// Mitsubishi GX Works2 project: testCode   PLC: FX3G

// global labels: Global1
VAR_GLOBAL
  Jog_Left AT X004 : BOOL;
  Jog_Right AT X006 : BOOL;
  RelayMXC_1 AT Y001 : BOOL;
  RelayMXC_2 AT Y002 : BOOL;
  CommandMXC_F : BOOL;
  CommandMXC_R : BOOL;
  MXC_FWD : BOOL;
  MXC_Z : BOOL;
END_VAR
VAR_GLOBAL CONSTANT
  Round_MXC : REAL := 2.5;
END_VAR
VAR_GLOBAL
  Real_MXC : REAL;
  ModeAuto : BOOL;
  HSC AT C238 : DINT;
END_VAR
VAR_GLOBAL CONSTANT
  Speed_MXC : REAL := 1.5;
END_VAR
VAR_GLOBAL
  Freq_MXC : REAL;
  Round_Int : DWORD;
  Freq_Int : DWORD;
END_VAR

// task Task_01 (event TRUE, interval 0, priority 31): Control
// task InterruptMXC_Z (event I401, interval 0, priority 31): PickupX004

PROGRAM Control
VAR
  MXC : MotorRev;
  FlashF : R_TRIG;
  FlashZ : F_TRIG;
  PushOilPump : BOOL;
  ButtonOilP : BOOL;
  FlashP : R_TRIG;
  CounterCK : INT;
  Servo_MXC : Servo;
END_VAR
(* Khai bao vong quay cho MXC*)
EI( TRUE );
DEMUL( TRUE, E2000.0, Round_MXC , Real_MXC);
DEMUL(TRUE, E48000.0, Speed_MXC, Freq_MXC);
DINT( TRUE ,  Real_MXC , Round_Int );
DINT( TRUE ,  Freq_MXC , Freq_Int );
(*
MXC(SetAutoMan:= ModeAuto,
			LimitInputF := MXC_FWD , LimitInputR := MXC_Z,
			SetAutoRunF := CommandMXC_F, SetAutoRunR := CommandMXC_R,
			OutputF := RelayMXC_1, OutputR := RelayMXC_2);

RST( LDF(TRUE, MXC_FWD), M8054);
SET( LDF(TRUE, MXC_FWD), MXC_Z);
SET( LDF(TRUE, MXC_FWD), CommandMXC_R);
SET( CommandMXC_F AND X004, MXC_FWD);
RST( LDP(TRUE, CommandMXC_F), C251);

OUT_C_32( TRUE, CC251, K2147483647);
DHSCR( TRUE , REAL_TO_DINT( Real_MXC ), CN251, MXC_FWD);
 *)


Servo_MXC(SetAutoMan := ModeAuto,
						LimitInputF:= MXC_FWD, LimitInputR:= MXC_Z,
						Speed:=  Round_Int, Range:= Freq_Int,
						SetAutoRunF:= CommandMXC_F , SetAutoRunR:= CommandMXC_R ,
						OutputPLS:= Y0, OutputDIR:= Y4 );

RST( LDF(TRUE, MXC_FWD), M8054);
SET( LDF(TRUE, MXC_FWD), MXC_Z);
SET( LDF(TRUE, MXC_FWD), CommandMXC_R);
SET( CommandMXC_F AND X004, MXC_FWD);
RST( LDF(TRUE, M8340), MXC_FWD);




ButtonOilP := LDP(TRUE, PushOilPump) XOR ButtonOilP;
END_PROGRAM

FUNCTION_BLOCK MotorRev
VAR_INPUT
  SetAutoMan : BOOL;
END_VAR
VAR_IN_OUT
  PushManF : BOOL;
  PushManR : BOOL;
END_VAR
VAR_INPUT
  LimitInputF : BOOL;
  LimitInputR : BOOL;
END_VAR
VAR_IN_OUT
  SetAutoRunF : BOOL;
  SetAutoRunR : BOOL;
END_VAR
VAR_OUTPUT
  OutputF : BOOL;
  OutputR : BOOL;
END_VAR
VAR
  RelayBufferF : BOOL;
  RelayBufferR : BOOL;
END_VAR
(* Set mode Auto/Man *)
IF  SetAutoMan THEN
	RelayBufferF := 	NOT SetAutoRunR AND SetAutoRunF;
	RelayBufferR := NOT SetAutoRunF AND SetAutoRunR;
ELSE
	RelayBufferF := NOT PushManR AND PushManF;
	RelayBufferR := NOT PushManF AND PushManR;
END_IF;

OutputF := RelayBufferF AND LimitInputF ;
OutputR := RelayBufferR AND LimitInputR ;
(* Reset control signal *)
RST( LDF( TRUE, LimitInputF ) , RelayBufferF );
RST( LDF( TRUE, LimitInputF ) , SetAutoRunF );

RST( LDF( TRUE, LimitInputR ) , RelayBufferR );	
RST( LDF( TRUE, LimitInputR ) , SetAutoRunR );
END_FUNCTION_BLOCK

PROGRAM PickupX004
RST( TRUE, MXC_Z);
SET( TRUE, M8054);
END_PROGRAM

FUNCTION_BLOCK Servo
VAR_INPUT
  SetAutoMan : BOOL;
  LimitInputF : BOOL;
  LimitInputR : BOOL;
END_VAR
VAR_IN_OUT
  PushManF : BOOL;
  PushManR : BOOL;
END_VAR
VAR_INPUT
  Speed : DWORD;
  Range : DWORD;
END_VAR
VAR_IN_OUT
  SetAutoRunF : BOOL;
  SetAutoRunR : BOOL;
END_VAR
VAR_OUTPUT
  OutputPLS : BOOL;
  OutputDIR : BOOL;
END_VAR
VAR
  RelayPLS : BOOL;
  RelayDIR : BOOL;
END_VAR
(* Set mode Auto/Man *)
IF  SetAutoMan THEN
	RelayDIR := SetAutoRunR;
	RelayPLS := SetAutoRunF XOR SetAutoRunR;
ELSE
	RelayDIR := PushManR;
	RelayPLS := PushManF XOR PushManR;
END_IF;

OutputDIR := RelayDIR ;

DPLSY( RelayPLS AND (LimitInputF OR LimitInputR) , Speed, Range , OutputPLS );

(* Reset control signal *)
RST( LDF( TRUE, LimitInputF ) , SetAutoRunF );
RST( LDF( TRUE, LimitInputR ) , SetAutoRunR );
END_FUNCTION_BLOCK
